Staubli VAL3: outputs.dtx

public dio bOut0 = {link=BasicIO-1\%Q0}
public dio bOut1 = {link=BasicIO-1\%Q1}
public dio bOut2 = {link=BasicIO-1\%Q2}
public dio bOut3 = {link=BasicIO-1\%Q3}
public dio bOut4 = {link=BasicIO-1\%Q4}
public dio bOut5 = {link=BasicIO-1\%Q5}
public dio bOut6 = {link=BasicIO-1\%Q6}
public dio bOut7 = {link=BasicIO-1\%Q7}
public dio bOut8 = {link=BasicIO-1\%Q8}
public dio bOut9 = {link=BasicIO-1\%Q9}
public dio bOut10 = {link=BasicIO-1\%Q10}
public dio bOut11 = {link=BasicIO-1\%Q11}
public dio bOut12 = {link=BasicIO-1\%Q12}
public dio bOut13 = {link=BasicIO-1\%Q13}
public dio bOut14 = {link=BasicIO-1\%Q14}
public dio bOut15 = {link=BasicIO-1\%Q15}
public dio b2Out0 = {link=BasicIO-2\%Q0}
public dio b2Out1 = {link=BasicIO-2\%Q1}
public dio b2Out2 = {link=BasicIO-2\%Q2}
public dio b2Out3 = {link=BasicIO-2\%Q3}
public dio b2Out4 = {link=BasicIO-2\%Q4}
public dio b2Out5 = {link=BasicIO-2\%Q5}
public dio b2Out6 = {link=BasicIO-2\%Q6}
public dio b2Out7 = {link=BasicIO-2\%Q7}
public dio b2Out8 = {link=BasicIO-2\%Q8}
public dio b2Out9 = {link=BasicIO-2\%Q9}
public dio b2Out10 = {link=BasicIO-2\%Q10}
public dio b2Out11 = {link=BasicIO-2\%Q11}
public dio b2Out12 = {link=BasicIO-2\%Q12}
public dio b2Out13 = {link=BasicIO-2\%Q13}
public dio b2Out14 = {link=BasicIO-2\%Q14}
public dio b2Out15 = {link=BasicIO-2\%Q15}
public dio cDout0 = {link=Can-Dio\%Q0}
public dio cDout1 = {link=Can-Dio\%Q1}
public dio cDout2 = {link=Can-Dio\%Q2}
public dio cDout3 = {link=Can-Dio\%Q3}
public dio cDout4 = {link=Can-Dio\%Q4}
public dio cDout5 = {link=Can-Dio\%Q5}
public dio cDout6 = {link=Can-Dio\%Q6}
public dio cDout7 = {link=Can-Dio\%Q7}
public dio fOut0 = {link=fOut0}
public dio mOut0 = {link=ModuleIO\%Q0}
public dio mOut1 = {link=ModuleIO\%Q1}
public dio mOut2 = {link=ModuleIO\%Q2}
public dio mOut3 = {link=ModbusSrv-0\Modbus-Bit\bOut3}
public dio mOut4 = {link=ModuleIO\%Q4}
public dio mOut5 = {link=ModuleIO\%Q5}
public dio mOut6 = {link=ModuleIO\%Q6}
public dio mOut7 = {link=ModuleIO\%Q7}
public dio mOut8 = {link=ModuleIO\%Q8}
public dio mOut9 = {link=ModuleIO\%Q9}
public dio mOut10 = {link=ModuleIO\%Q10}
public dio mOut11 = {link=ModuleIO\%Q11}
public dio mOut12 = {link=ModuleIO\%Q12}
public dio mOut13 = {link=ModuleIO\%Q13}
public dio mOut14 = {link=ModuleIO\%Q14}
public dio mOut15 = {link=ModuleIO\%Q15}
public dio mOut16 = {link=ModuleIO\%Q16}
public dio mOut17 = {link=ModuleIO\%Q17}
public dio mOut18 = {link=ModuleIO\%Q18}
public dio mOut19 = {link=ModuleIO\%Q19}
public dio mOut20 = {link=ModuleIO\%Q20}
public dio mOut21 = {link=ModuleIO\%Q21}
public dio mOut22 = {link=ModuleIO\%Q22}
public dio mOut23 = {link=ModuleIO\%Q23}
public dio mOut24 = {link=ModuleIO\%Q24}
public dio mOut25 = {link=ModuleIO\%Q25}
public dio mOut26 = {link=ModuleIO\%Q26}
public dio mOut27 = {link=ModuleIO\%Q27}
public dio mOut28 = {link=ModuleIO\%Q28}
public dio mOut29 = {link=ModuleIO\%Q29}
public dio mOut30 = {link=ModuleIO\%Q30}
public dio mOut31 = {link=ModuleIO\%Q31}
